SUBAPPLICATION Uebung_221b_ALR (* Standard IEC 61131-3 ADI_FB_CTUD (Adapter Version, Vorwärts-/Rückwärtszähler, DINT) mit Terminal-Ausgabe (PHYS) *)
  (* Standard: 61131-3; Description: Copyright (c) 2026 Meisterschulen am Ostbahnhof This program and the accompanying materials are made available under the terms of the Eclipse Public License 2.0 which is available at https://www.eclipse.org/legal/epl-2.0/ SPDX-License-Identifier: EPL-2.0 *)
  (* Version 1.2, 2026-05-13, Franz Höpfinger, Meisterschulen am Ostbahnhof, Added ADI_DINT_TO_DI init block connected to PV *)
  (* Version 1.1, 2026-04-21, Franz Höpfinger, Meisterschulen am Ostbahnhof, Added terminal output for counter value (PHYS) *)
  (* Version 1.0, 2026-04-21, Franz Höpfinger, Meisterschulen am Ostbahnhof, initial API and implementation (Adapter version) *)
  PACKAGE Uebungen;
  IMPORT Uebungen::const::UT::DefaultPool_Numeric::OutputNumber_N3_N;
  IMPORT logiBUS::io::DI::logiBUS_DI::Input_I1;
  IMPORT logiBUS::io::DI::logiBUS_DI::Input_I2;
  IMPORT logiBUS::io::DI::logiBUS_DI::Input_I3;
  IMPORT logiBUS::io::DI::logiBUS_DI::Input_I4;
  IMPORT logiBUS::io::DQ::logiBUS_DO::Output_Q1;
  IMPORT logiBUS::io::DQ::logiBUS_DO::Output_Q2;
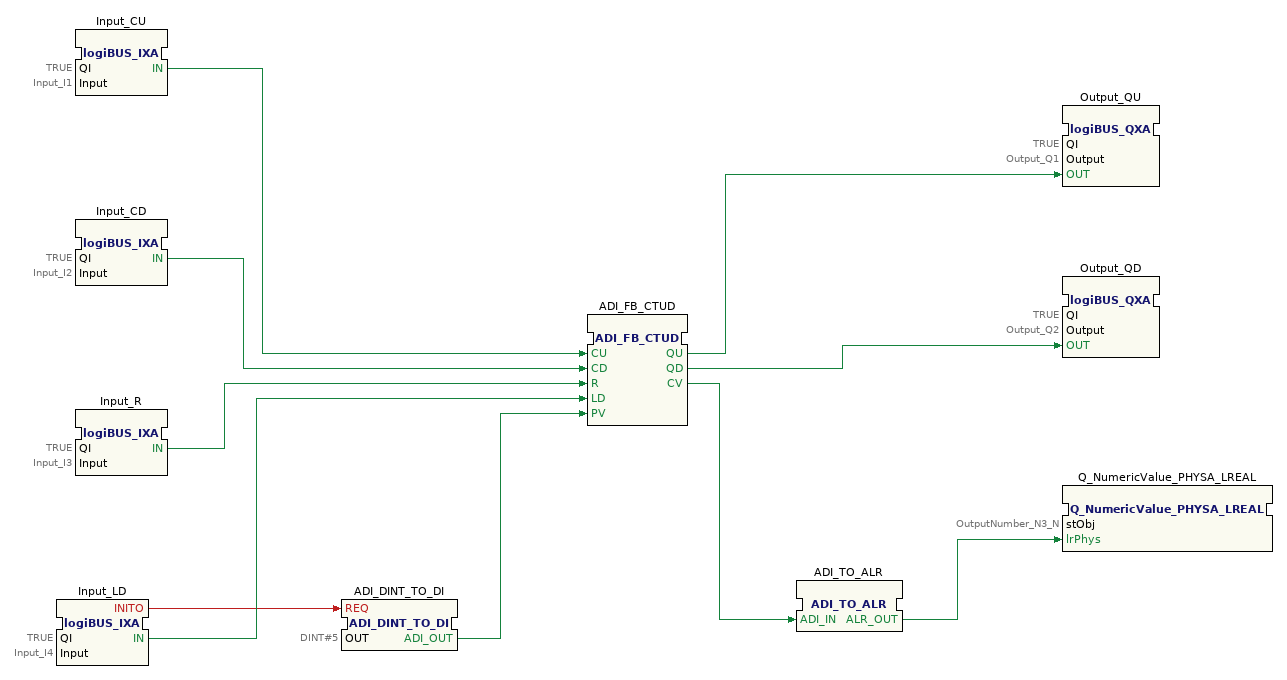
  (* hier sind negative Werte möglich ! *)
  (* hier gegebenenfalls je einen AX_D_FF einbauen, damit die Events reduziert werden. *)
  FBS
    ADI_FB_CTUD : adapter::iec61131::counters::ADI_FB_CTUD;
    ADI_DINT_TO_DI : adapter::conversion::unidirectional::ADI_DINT_TO_DI(OUT := DINT#5);
    Input_CU : logiBUS::io::DI::logiBUS_IXA(QI := TRUE, Input := Input_I1);
    Input_CD : logiBUS::io::DI::logiBUS_IXA(QI := TRUE, Input := Input_I2);
    Input_R : logiBUS::io::DI::logiBUS_IXA(QI := TRUE, Input := Input_I3);
    Input_LD : logiBUS::io::DI::logiBUS_IXA(QI := TRUE, Input := Input_I4);
    Output_QU : logiBUS::io::DQ::logiBUS_QXA(QI := TRUE, Output := Output_Q1);
    Output_QD : logiBUS::io::DQ::logiBUS_QXA(QI := TRUE, Output := Output_Q2);
    ADI_TO_ALR : adapter::conversion::unidirectional::ADI_TO_ALR;
    Q_NumericValue_PHYSA_LREAL : isobus::UT::Q::Q_NumericValue_PHYSA_LREAL(stObj := OutputNumber_N3_N);
  END_FBS
  EVENT_CONNECTIONS
    Input_LD.INITO TO ADI_DINT_TO_DI.REQ;
  END_CONNECTIONS
  ADAPTER_CONNECTIONS
    Input_CU.IN TO ADI_FB_CTUD.CU;
    Input_CD.IN TO ADI_FB_CTUD.CD;
    Input_R.IN TO ADI_FB_CTUD.R;
    Input_LD.IN TO ADI_FB_CTUD.LD;
    ADI_FB_CTUD.QU TO Output_QU.OUT;
    ADI_FB_CTUD.QD TO Output_QD.OUT;
    ADI_FB_CTUD.CV TO ADI_TO_ALR.ADI_IN;
    ADI_TO_ALR.ALR_OUT TO Q_NumericValue_PHYSA_LREAL.lrPhys;
    ADI_DINT_TO_DI.ADI_OUT TO ADI_FB_CTUD.PV;
  END_CONNECTIONS
END_SUBAPPLICATION
